// TwinCAT 3 PLC project TEST
// ProgramVersion: 3.1.4026.11
// libraries:
//   Tc2_ModbusRTU, * (Beckhoff Automation GmbH)
//   Tc2_ModbusSrv, * (Beckhoff Automation GmbH)
//   Tc2_Standard, * (Beckhoff Automation GmbH)
//   Tc2_System, * (Beckhoff Automation GmbH)
// project tree:
//   GVLs/ GVL_HMI.TcGVL, GVL_Simulated.TcGVL
//   / PlcTask.TcTTO
//   POUs/ AssignInsOuts.TcPOU, HMI_Functions.TcPOU, MAIN.TcPOU, Part1.TcPOU, Part2.TcPOU, Part3.TcPOU
//   POUs/Function Blocks/ FB_FactoryIO_ReadInputs_.TcPOU, FB_FactoryIO_WriteOutputs.TcPOU
// real-time tasks:
//   TASK Device 1 (OPC UA Virtual)_Task_58: cycle T#40ms, priority 58, ADS port 350
//   TASK PlcTask: cycle T#10ms, priority 20, ADS port 351
//   TASK PlcTask1: cycle T#10ms, priority 21, ADS port 352

CONFIGURATION TEST
    RESOURCE PLC ON TwinCAT3
        TASK PlcTask(INTERVAL := T#10ms, PRIORITY := 20);
        PROGRAM MAIN WITH PlcTask : MAIN;
    END_RESOURCE
END_CONFIGURATION

// ---- GVLs/GVL_HMI.TcGVL
{attribute 'qualified_only'}
VAR_GLOBAL
	b_StartAuto : BOOL;
	b_StopAuto : BOOL;
	ProgramSelect : DINT;
END_VAR

// ---- GVLs/GVL_Simulated.TcGVL
{attribute 'qualified_only'}
VAR_GLOBAL
	//FIO Inputs
	b_Sensor1 : BOOL;
	b_Sensor2 : BOOL;
	b_Sensor3 : BOOL;
	b_Sensor4 : BOOL;
	b_Sensor2_1 : BOOL;
	b_Sensor2_2 : BOOL;
	b_Sensor2_3 : BOOL;
//FIO Outputs
	b_ConvPos : BOOL;
	b_ConvNeg : BOOL;
	b_Light1 : BOOL;
	b_Light2 : BOOL;
	b_Light3 : BOOL;
	b_Light4 : BOOL;
	b_conv2_1 : BOOL;
	b_conv2_2 : BOOL;
	b_conv2_3 : BOOL;
	b_Emitter : BOOL;
	b_Remover : BOOL;
END_VAR

// ---- POUs/MAIN.TcPOU
PROGRAM MAIN
VAR

END_VAR


AssignInsOuts();

HMI_Functions();

CASE GVL_HMI.ProgramSelect OF
	1:
		Part1();
	2:
		Part2();
	3:
		Part3();
END_CASE

END_PROGRAM

// ---- POUs/AssignInsOuts.TcPOU
PROGRAM AssignInsOuts
VAR
	//Factory IO
	FactoryIO_Ins : ARRAY [0..15] OF BYTE;
	FactoryIO_Outs : ARRAY [0..15] OF BYTE;
	FactoryIO_RegOuts : ARRAY [0..7] OF BYTE;
	
	//FIO Function Blocks
	FB_FactoryIO_ReadInputs: FB_FactoryIO_ReadInputs_;
	FB_FactoryIO_WriteOutputs: FB_FactoryIO_WriteOutputs;
END_VAR

//Reads Inputs and Writes Outputs to FactoryIO over TCP/IP
FB_FactoryIO_ReadInputs();
FB_FactoryIO_WriteOutputs();


//Link Inputs from FactoryIO
GVL_Simulated.b_Sensor1 := NOT FactoryIO_Ins [0].0;
GVL_Simulated.b_Sensor2 := NOT FactoryIO_Ins [0].1;
GVL_Simulated.b_Sensor3 := NOT FactoryIO_Ins [0].2;
GVL_Simulated.b_Sensor4 := NOT FactoryIO_Ins [0].3;
GVL_Simulated.b_Sensor2_1 := NOT FactoryIO_Ins [0].4;
GVL_Simulated.b_Sensor2_2 := NOT FactoryIO_Ins [0].5;
GVL_Simulated.b_Sensor2_3 := NOT FactoryIO_Ins [0].6;


//Link Outputs to FactoryIO
FactoryIO_Outs [0].0 := GVL_Simulated.b_convPos ;
FactoryIO_Outs [0].1 := GVL_Simulated.b_convNeg ;
FactoryIO_Outs [0].2 := GVL_Simulated.b_light1 ;
FactoryIO_Outs [0].3 := GVL_Simulated.b_light2 ;
FactoryIO_Outs [0].4 := GVL_Simulated.b_light3 ;
FactoryIO_Outs [0].5 := GVL_Simulated.b_light4 ;
FactoryIO_Outs [0].6 := GVL_Simulated.b_conv2_1 ;
FactoryIO_Outs [0].7 := GVL_Simulated.b_conv2_2 ;
FactoryIO_Outs [1].0 := GVL_Simulated.b_conv2_3 ;
FactoryIO_Outs [1].1 := GVL_Simulated.b_Emitter ;
FactoryIO_Outs [1].2 := GVL_Simulated.b_Remover ;

END_PROGRAM

// ---- POUs/Function Blocks/FB_FactoryIO_ReadInputs_.TcPOU
FUNCTION_BLOCK FB_FactoryIO_ReadInputs_
VAR_INPUT
END_VAR
VAR_OUTPUT
END_VAR
VAR
	FactoryIO_ReadInsFB : FB_MBReadInputs;
	
END_VAR

FactoryIO_ReadInsFB(
	sIPAddr:= '127.0.0.1' , 
	nTCPPort:= 75, 
	nUnitID:= 1, 
	nQuantity:= 16, 
	nMBAddr:= 0, 
	cbLength:= SIZEOF(AssignInsOuts.FactoryIO_Ins), 
	pDestAddr:= ADR(AssignInsOuts.FactoryIO_Ins), 
	bExecute:= TRUE, 
	tTimeout:= T#1S, 
	bBusy=> , 
	bError=> , 
	nErrId=> , 
	cbRead=> );

FactoryIO_ReadInsFB(bExecute:=FALSE);

END_FUNCTION_BLOCK

// ---- POUs/Function Blocks/FB_FactoryIO_WriteOutputs.TcPOU
FUNCTION_BLOCK FB_FactoryIO_WriteOutputs
VAR_INPUT
END_VAR
VAR_OUTPUT
END_VAR
VAR
	FactoryIO_WriteOutsFB : FB_MBWriteCoils;
END_VAR

FactoryIO_WriteOutsFB(
	sIPAddr:= '127.0.0.1', 
	nTCPPort:= 75, 
	nUnitID:= 1, 
	nQuantity:= 16, 
	nMBAddr:= 0, 
	cbLength:= SIZEOF(AssignInsOuts.FactoryIO_Outs), 
	pSrcAddr:= ADR(AssignInsOuts.FactoryIO_Outs), 
	bExecute:= TRUE, 
	tTimeout:= T#1S, 
	bBusy=> , 
	bError=> , 
	nErrId=> );
	
	FactoryIO_WriteOutsFB(bExecute:=FALSE);

END_FUNCTION_BLOCK

// ---- POUs/HMI_Functions.TcPOU
PROGRAM HMI_Functions
VAR
	PointLeft : STRING := 'Visible';
	PointRight : STRING := 'Visible';
	RightBox : STRING := 'Visible';
	LeftBox : STRING := 'Visible';
	
END_VAR


//Programs Box direction layout on HMI Control Screen
CASE Part1.ProcessState OF
	0://MachineStop
		PointLeft := 'Hidden';
		PointRight := 'Hidden';
		RightBox := 'Hidden';
		LeftBox := 'Hidden';
	1://Positive Direction
		PointLeft := 'Hidden';
		PointRight := 'Visible';
		RightBox := 'Hidden';
		LeftBox := 'Hidden';
	2://Hold
		PointLeft := 'Hidden';
		PointRight := 'Hidden';
		RightBox := 'Visible';
		LeftBox := 'Hidden';
	3://Negative Direction
		PointLeft := 'Visible';
		PointRight := 'Hidden';
		RightBox := 'Hidden';
		LeftBox := 'Hidden';
	4://Hold
		PointLeft := 'Hidden';
		PointRight := 'Hidden';
		RightBox := 'Hidden';
		LeftBox := 'Visible';
	
END_CASE

END_PROGRAM

// ---- POUs/Part1.TcPOU
PROGRAM Part1
VAR
//Program Components
	ProcessState : INT := 0;
	CycleTrack : INT :=0;
	HoldTime : TON;
	ProcessStopped: BOOL;
END_VAR

HoldTime(PT := T#1S );




IF GVL_HMI.b_StopAuto THEN
	ProcessStopped := TRUE;
END_IF

IF ProcessStopped THEN
	GVL_Simulated.b_ConvPos := GVL_Simulated.b_ConvNeg := FALSE;
	HoldTime.IN := FALSE;
END_IF

IF GVL_HMI.b_StartAuto THEN
	ProcessStopped := FALSE;
END_IF


IF NOT ProcessStopped THEN
	CASE ProcessState OF
		0://MachineStop
			GVL_Simulated.b_ConvPos := GVL_Simulated.b_ConvNeg := FALSE;
			IF GVL_HMI.b_StartAuto THEN
				ProcessState :=1;
			END_IF
		1://Positive Direction
			GVL_Simulated.b_ConvPos := TRUE;
			GVL_Simulated.b_ConvNeg := FALSE;
			IF GVL_Simulated.b_Sensor4 THEN
				ProcessState :=2;
				CycleTrack := CycleTrack +1;
			END_IF
		2://Hold
			GVL_Simulated.b_ConvPos := GVL_Simulated.b_ConvNeg := FALSE;
			HoldTime.IN := TRUE;
			IF HoldTime.Q THEN
				HoldTime.IN := FALSE;
				ProcessState :=3;
			END_IF
		3://Negative Direction
			GVL_Simulated.b_ConvNeg := TRUE;
			GVL_Simulated.b_ConvPos := FALSE;
			IF GVL_Simulated.b_Sensor1 THEN
				ProcessState :=4;
				CycleTrack := CycleTrack +1;
			END_IF
		4://Hold
			GVL_Simulated.b_ConvPos := GVL_Simulated.b_ConvNeg := FALSE;
			HoldTime.IN := TRUE;
			IF HoldTime.Q THEN
				HoldTime.IN := FALSE;
				ProcessState :=1;
			END_IF
		
	END_CASE
END_IF


IF CycleTrack = 21 THEN
	ProcessState := 0;
END_IF

END_PROGRAM

// ---- POUs/Part2.TcPOU
PROGRAM Part2
VAR
	//Program Components
	ProcessState : INT := 0;
	CycleTrack : INT :=0;
	HoldTime : TON;
	ProcessStopped: BOOL := False;
END_VAR

//Initialize Hold Timer
HoldTime(PT := T#3S );

//Set Lights and Motors to Default Off
gvl_simulated.b_Light1 := gvl_simulated.b_Light2 :=gvl_simulated.b_Light3 :=gvl_simulated.b_Light4 := FALSE;
GVL_Simulated.b_ConvPos := GVL_Simulated.b_ConvNeg := FALSE;

//Detects if Stop Button Pressed
IF GVL_HMI.b_StopAuto THEN
	ProcessStopped := TRUE;
END_IF
IF ProcessStopped THEN
	HoldTime.IN := FALSE;
END_IF
IF GVL_HMI.b_StartAuto THEN
	ProcessStopped := FALSE;
END_IF

//State Machine
IF NOT ProcessStopped THEN
	CASE ProcessState OF
		
		0://MachineStop
			IF GVL_HMI.b_StartAuto THEN
				ProcessState :=1;
			END_IF
			
		1://1 to 2
			GVL_Simulated.b_ConvPos := TRUE;
			IF GVL_Simulated.b_Sensor2 THEN
				ProcessState :=2;
				CycleTrack := CycleTrack +1;
			END_IF
			
		2://Hold 2
			gvl_simulated.b_Light2 := TRUE;
			HoldTime.IN := TRUE;
			IF HoldTime.Q THEN
				HoldTime.IN := FALSE;
				ProcessState :=3;
			END_IF
			
		3://2 to 3
			GVL_Simulated.b_ConvPos := TRUE;
			IF GVL_Simulated.b_Sensor3 THEN
				ProcessState :=4;
				CycleTrack := CycleTrack +1;
			END_IF
			
		4://Hold 3
			gvl_simulated.b_Light3 := TRUE;
			HoldTime.IN := TRUE;
			IF HoldTime.Q THEN
				HoldTime.IN := FALSE;
				ProcessState :=5;
			END_IF
			
		5://3 to 4
			GVL_Simulated.b_ConvPos := TRUE;
			IF GVL_Simulated.b_Sensor4 THEN
				ProcessState :=6;
				CycleTrack := CycleTrack +1;
			END_IF
			
		6://Hold 4
			HoldTime.IN := TRUE;
			gvl_simulated.b_Light4 := TRUE;
			IF HoldTime.Q THEN
				HoldTime.IN := FALSE;
				ProcessState :=7;
			END_IF
			
		7://4 to 3
			GVL_Simulated.b_ConvNeg := TRUE;
			IF GVL_Simulated.b_Sensor3 THEN
				ProcessState :=8;
				CycleTrack := CycleTrack +1;
			END_IF
			
		8://Hold 3
			HoldTime.IN := TRUE;
			gvl_simulated.b_Light3 := TRUE;
			IF HoldTime.Q THEN
				HoldTime.IN := FALSE;
				ProcessState :=9;
			END_IF
			
		9://3 to 2
			GVL_Simulated.b_ConvNeg := TRUE;
			IF GVL_Simulated.b_Sensor2 THEN
				ProcessState :=10;
				CycleTrack := CycleTrack +1;
			END_IF
			
		10://Hold 2
			HoldTime.IN := TRUE;
			gvl_simulated.b_Light2 := TRUE;
			IF HoldTime.Q THEN
				HoldTime.IN := FALSE;
				ProcessState :=11;
			END_IF
			
		11://2 to 1
			GVL_Simulated.b_ConvNeg := TRUE;
			IF GVL_Simulated.b_Sensor1 THEN
				ProcessState :=12;
				CycleTrack := CycleTrack +1;
			END_IF
			
		12://Hold 1
			HoldTime.IN := TRUE;
			gvl_simulated.b_Light1 := TRUE;
			IF HoldTime.Q THEN
				HoldTime.IN := FALSE;
				ProcessState :=1;
			END_IF
			
	END_CASE
	
END_IF



(*
IF CycleTrack = 21 THEN
	ProcessState := 0;
END_IF
*)

END_PROGRAM

// ---- POUs/Part3.TcPOU
PROGRAM Part3
VAR
//Program Components
	ProcessState : INT := 0;
	ProcessStopped: BOOL := FALSE;
END_VAR



//Set Lights and Motors to Default Off
GVL_Simulated.b_Emitter := GVL_Simulated.b_Remover := FALSE;
GVL_Simulated.b_conv2_1 := GVL_Simulated.b_conv2_2 := GVL_Simulated.b_conv2_3 := FALSE;

//Detects if Stop Button Pressed
IF GVL_HMI.b_StopAuto THEN
	ProcessStopped := TRUE;
END_IF

IF GVL_HMI.b_StartAuto THEN
	ProcessStopped := FALSE;
END_IF

//State Machine
IF NOT ProcessStopped THEN
	CASE ProcessState OF
		
		0://Process Start
			IF GVL_HMI.b_StartAuto THEN
				ProcessState :=10;
			END_IF
		10:// Emit
			GVL_Simulated.b_Emitter := TRUE;
			IF  GVL_Simulated.b_Sensor2_1 THEN
				ProcessState :=20;
			END_IF
			
		20://1 to 2
			GVL_Simulated.b_conv2_1 := TRUE;
			GVL_Simulated.b_conv2_2 := TRUE;
			IF GVL_Simulated.b_Sensor2_2 THEN
				ProcessState :=30;
			END_IF

		30://2 to 3
			GVL_Simulated.b_conv2_2 := TRUE;
			GVL_Simulated.b_conv2_3 := TRUE;
			IF GVL_Simulated.b_Sensor2_3 THEN
				ProcessState :=40;
			END_IF
			
			
		40://3 to 4
			GVL_Simulated.b_conv2_3 := TRUE;
			IF GVL_Simulated.b_Sensor2_3 THEN
				ProcessState :=50;
			END_IF
		50: //Remove Items
			GVL_Simulated.b_Remover := TRUE;
			IF NOT GVL_Simulated.b_Sensor2_3 THEN
				ProcessState :=10;
			END_IF
	END_CASE
END_IF

END_PROGRAM
